Fanuc KAREL source: kt00192.KL

-- PROVISIONAL review KL for V770-1; original PC SHA256 dda5013808225450db4fcf76ae9d8ff175c5f036ea0b959ca5c4380af92a72a5
-- Incomplete behavior may be omitted. Consult companion uncertainty JSON. Do not deploy.
PROGRAM KT00192
%NOLOCKGROUP
VAR
  OUT : REAL
-- UNRESOLVED_DECL H1 type=002017
-- UNRESOLVED_DECL H2 type=002017
BEGIN
  -- UNRESOLVED_PC offsets 5-19; opcodes 2E,22,9D,33,B4
  -- UNRESOLVED_PC offsets 24-38; opcodes 2E,22,9D,33,B4
  -- UNRESOLVED_PC offsets 43-57; opcodes 2E,22,9D,33,B4
  -- UNRESOLVED_PC offsets 62-76; opcodes 2E,22,9D,33,B4
  -- UNRESOLVED_PC offsets 81-107; opcodes 22,9D,33,B3,22,9D,33,B3,56,64,23
  -- UNRESOLVED_PC offsets 112-116; opcodes 7F
END KT00192
